// TIA Portal V15.1 export
// export: Created 2024-06-21T08:40:52.1288685Z, ExportSetting WithDefaults, DisplayName Totally Integrated Automation Portal, DisplayVersion V15.1 Update 5, DisplayName TIA Portal Openness, DisplayVersion V15.1 Update 5, DisplayName SINAMICS Startdrive Advanced, DisplayVersion V15.1, DisplayName G130, G150, S120, S150, SINAMICS MV, S210, DisplayVersion V15.1, DisplayName G110M, G120, G120C, G120D, G120P, DisplayVersion V15.1, DisplayName STEP 7 Professional, DisplayVersion V15.1 Update 5, DisplayName STEP 7 Safety, DisplayVersion V15.1, DisplayName WinCC Professional, DisplayVersion V15.1 Update 5, DisplayName SIMATIC Visualization Architect, DisplayVersion V15.1
FUNCTION "F209210ZS01Output" : Void   // FC7012, F_FBD
TITLE = Safety Inputs ZMProc / Safety Outputs 209210ZS01
{ S7_Optimized_Access := 'TRUE' }
VERSION : 0.1
// stored: AutoNumber false, IsIECCheckEnabled false, UDAEnableTagReadback false
BEGIN

REGION Network 1: **** --------------------- Infeed Roller // 210CR21 --------------------- ****
END_REGION

REGION Network 2: **** 8 - Outputs **** 209000AK03M1-UE130 Power OFF - 210CR21M1
   // SEW Drive Power OFF
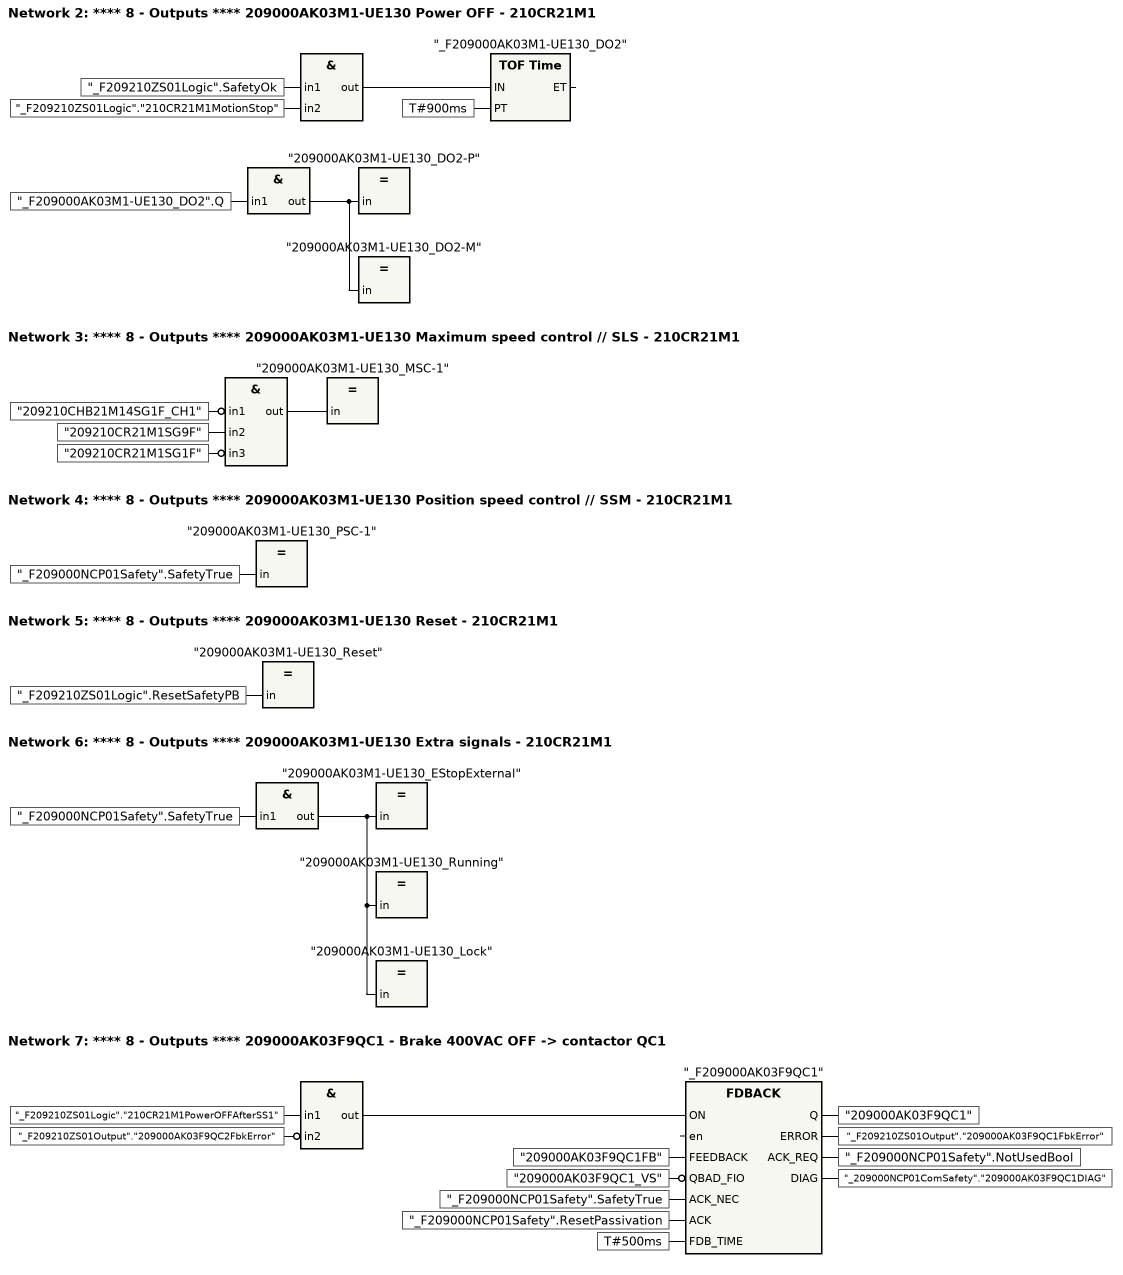
   "_F209000AK03M1-UE130_DO2".TOF(IN := "_F209210ZS01Logic".SafetyOk AND "_F209210ZS01Logic"."210CR21M1MotionStop",
                           PT := T#900ms);
   "209000AK03M1-UE130_DO2-P" := "_F209000AK03M1-UE130_DO2".Q;
   "209000AK03M1-UE130_DO2-M" := "_F209000AK03M1-UE130_DO2".Q;
END_REGION

REGION Network 3: **** 8 - Outputs **** 209000AK03M1-UE130 Maximum speed control // SLS - 210CR21M1
   // SEW Drive Maximum speed control
   "209000AK03M1-UE130_MSC-1" := NOT "209210CHB21M14SG1F_CH1" AND "209210CR21M1SG9F" AND NOT "209210CR21M1SG1F";
END_REGION

REGION Network 4: **** 8 - Outputs **** 209000AK03M1-UE130 Position speed control // SSM - 210CR21M1
   "209000AK03M1-UE130_PSC-1" := "_F209000NCP01Safety".SafetyTrue;
END_REGION

REGION Network 5: **** 8 - Outputs **** 209000AK03M1-UE130 Reset - 210CR21M1
   // SEW Drive Reset
   "209000AK03M1-UE130_Reset" := "_F209210ZS01Logic".ResetSafetyPB;
END_REGION

REGION Network 6: **** 8 - Outputs **** 209000AK03M1-UE130 Extra signals - 210CR21M1
   // SEW Drive Extra signals
   "209000AK03M1-UE130_EStopExternal" := "_F209000NCP01Safety".SafetyTrue;
   "209000AK03M1-UE130_Running" := "_F209000NCP01Safety".SafetyTrue;
   "209000AK03M1-UE130_Lock" := "_F209000NCP01Safety".SafetyTrue;
END_REGION

REGION Network 7: **** 8 - Outputs **** 209000AK03F9QC1 - Brake 400VAC OFF -> contactor QC1
   // Brake 400VAC OFF
   "_F209000AK03F9QC1"(ON := "_F209210ZS01Logic"."210CR21M1PowerOFFAfterSS1" AND NOT "_F209210ZS01Output"."209000AK03F9QC2FbkError",   // FDBACK
                       FEEDBACK := "209000AK03F9QC1FB",
                       QBAD_FIO := NOT "209000AK03F9QC1_VS",
                       ACK_NEC := "_F209000NCP01Safety".SafetyTrue,
                       ACK := "_F209000NCP01Safety".ResetPassivation,
                       FDB_TIME := T#500ms,
                       Q => "209000AK03F9QC1",
                       ERROR => "_F209210ZS01Output"."209000AK03F9QC1FbkError",
                       ACK_REQ => "_F209000NCP01Safety".NotUsedBool,
                       DIAG => "_209000NCP01ComSafety"."209000AK03F9QC1DIAG");
END_REGION

REGION Network 8: **** 8 - Outputs **** 209000AK03F9QC2 - Brake 400VAC OFF -> contactor QC2
   // Brake 400VAC OFF
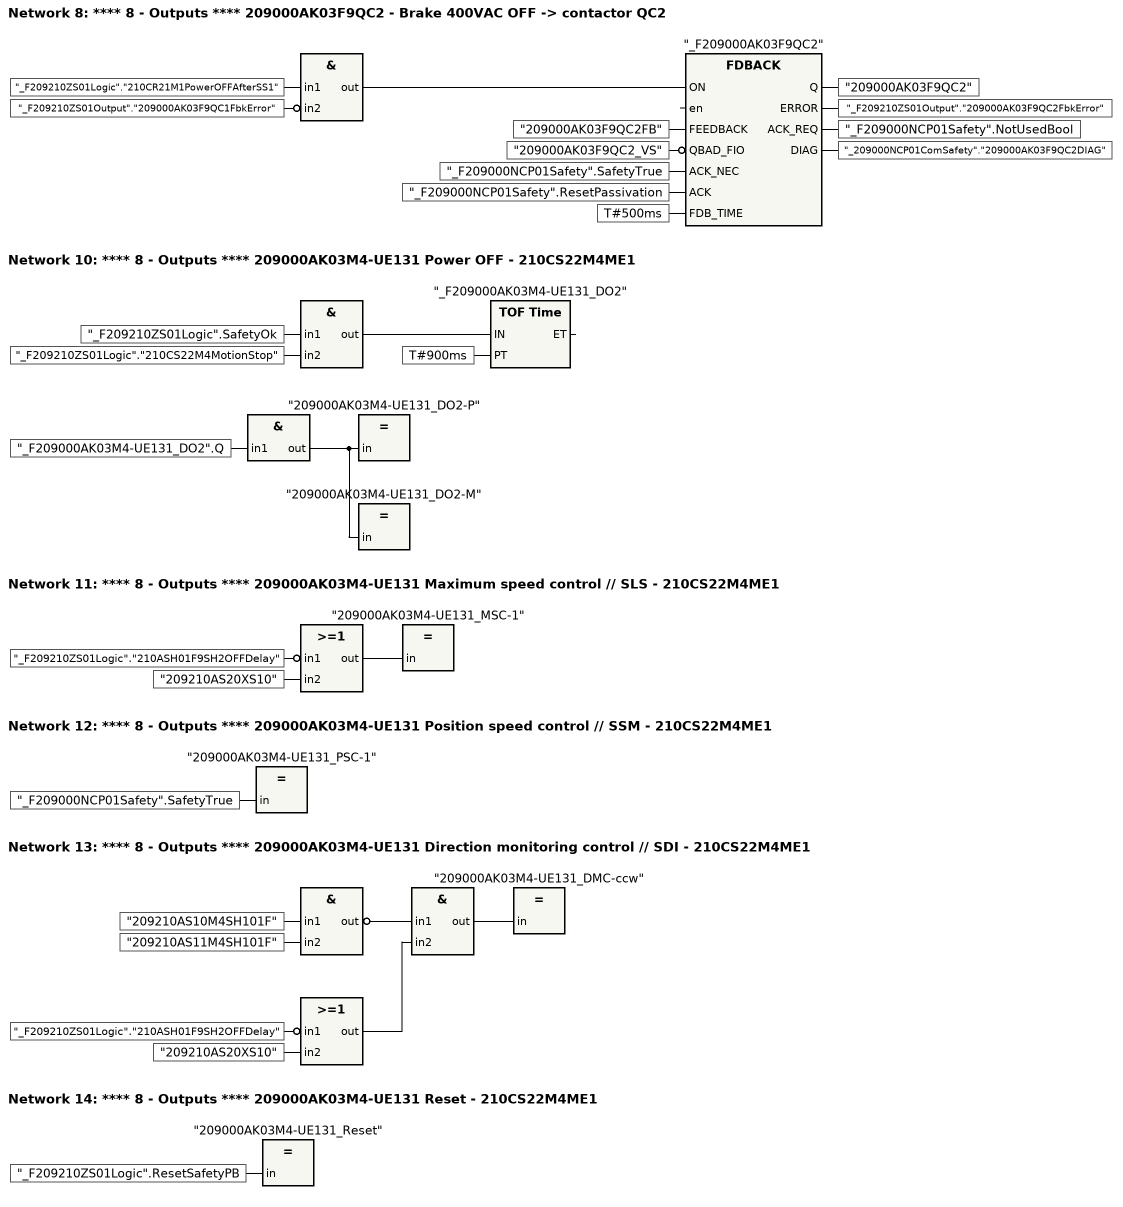
   "_F209000AK03F9QC2"(ON := "_F209210ZS01Logic"."210CR21M1PowerOFFAfterSS1" AND NOT "_F209210ZS01Output"."209000AK03F9QC1FbkError",   // FDBACK
                       FEEDBACK := "209000AK03F9QC2FB",
                       QBAD_FIO := NOT "209000AK03F9QC2_VS",
                       ACK_NEC := "_F209000NCP01Safety".SafetyTrue,
                       ACK := "_F209000NCP01Safety".ResetPassivation,
                       FDB_TIME := T#500ms,
                       Q => "209000AK03F9QC2",
                       ERROR => "_F209210ZS01Output"."209000AK03F9QC2FbkError",
                       ACK_REQ => "_F209000NCP01Safety".NotUsedBool,
                       DIAG => "_209000NCP01ComSafety"."209000AK03F9QC2DIAG");
END_REGION

REGION Network 9: **** --------------------- Slat Conveyor // 210CS22 --------------------- ****
END_REGION

REGION Network 10: **** 8 - Outputs **** 209000AK03M4-UE131 Power OFF - 210CS22M4ME1
   // SEW Drive Power OFF
   "_F209000AK03M4-UE131_DO2".TOF(IN := "_F209210ZS01Logic".SafetyOk AND "_F209210ZS01Logic"."210CS22M4MotionStop",
                           PT := T#900ms);
   "209000AK03M4-UE131_DO2-P" := "_F209000AK03M4-UE131_DO2".Q;
   "209000AK03M4-UE131_DO2-M" := "_F209000AK03M4-UE131_DO2".Q;
END_REGION

REGION Network 11: **** 8 - Outputs **** 209000AK03M4-UE131 Maximum speed control // SLS - 210CS22M4ME1
   // SEW Drive Maximum speed control
   "209000AK03M4-UE131_MSC-1" := NOT "_F209210ZS01Logic"."210ASH01F9SH2OFFDelay" OR "209210AS20XS10";
END_REGION

REGION Network 12: **** 8 - Outputs **** 209000AK03M4-UE131 Position speed control // SSM - 210CS22M4ME1
   "209000AK03M4-UE131_PSC-1" := "_F209000NCP01Safety".SafetyTrue;
END_REGION

REGION Network 13: **** 8 - Outputs **** 209000AK03M4-UE131 Direction monitoring control // SDI - 210CS22M4ME1
   "209000AK03M4-UE131_DMC-ccw" := NOT ("209210AS10M4SH101F" AND "209210AS11M4SH101F") AND (NOT "_F209210ZS01Logic"."210ASH01F9SH2OFFDelay" OR "209210AS20XS10");
END_REGION

REGION Network 14: **** 8 - Outputs **** 209000AK03M4-UE131 Reset - 210CS22M4ME1
   // SEW Drive Reset
   "209000AK03M4-UE131_Reset" := "_F209210ZS01Logic".ResetSafetyPB;
END_REGION

REGION Network 15: **** 8 - Outputs **** 209000AK03M4-UE131 Extra signals - 210CS22M4ME1
   // SEW Drive Extra signals
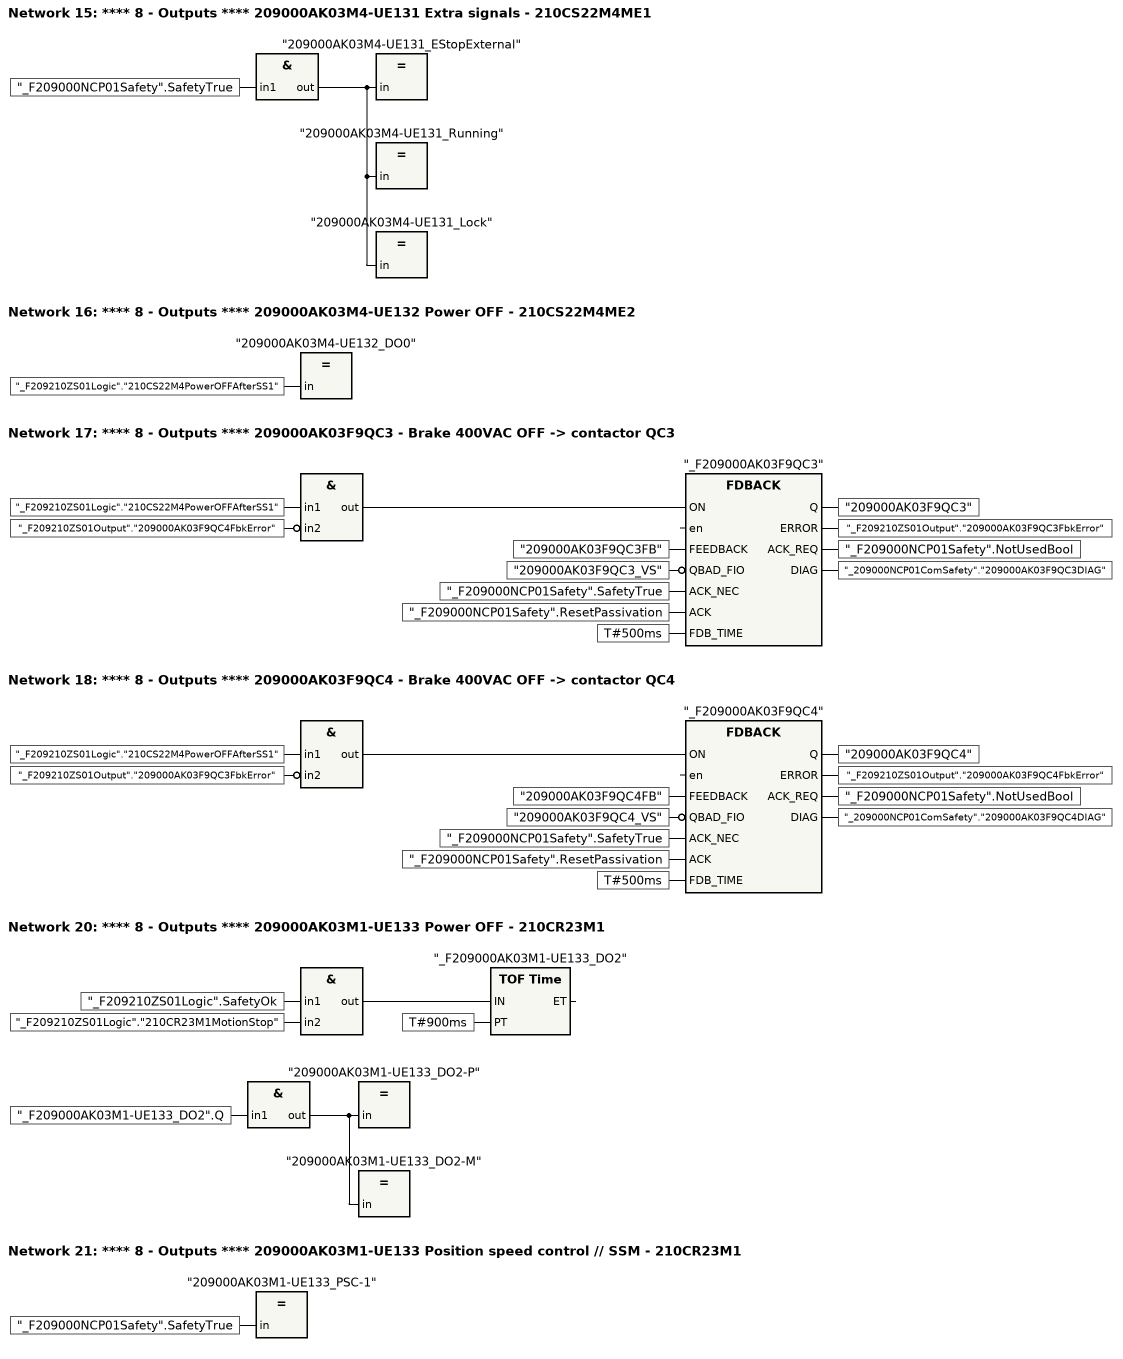
   "209000AK03M4-UE131_EStopExternal" := "_F209000NCP01Safety".SafetyTrue;
   "209000AK03M4-UE131_Running" := "_F209000NCP01Safety".SafetyTrue;
   "209000AK03M4-UE131_Lock" := "_F209000NCP01Safety".SafetyTrue;
END_REGION

REGION Network 16: **** 8 - Outputs **** 209000AK03M4-UE132 Power OFF - 210CS22M4ME2
   // SEW Drive Power OFF
   "209000AK03M4-UE132_DO0" := "_F209210ZS01Logic"."210CS22M4PowerOFFAfterSS1";
END_REGION

REGION Network 17: **** 8 - Outputs **** 209000AK03F9QC3 - Brake 400VAC OFF -> contactor QC3
   // Brake 400VAC OFF
   "_F209000AK03F9QC3"(ON := "_F209210ZS01Logic"."210CS22M4PowerOFFAfterSS1" AND NOT "_F209210ZS01Output"."209000AK03F9QC4FbkError",   // FDBACK
                       FEEDBACK := "209000AK03F9QC3FB",
                       QBAD_FIO := NOT "209000AK03F9QC3_VS",
                       ACK_NEC := "_F209000NCP01Safety".SafetyTrue,
                       ACK := "_F209000NCP01Safety".ResetPassivation,
                       FDB_TIME := T#500ms,
                       Q => "209000AK03F9QC3",
                       ERROR => "_F209210ZS01Output"."209000AK03F9QC3FbkError",
                       ACK_REQ => "_F209000NCP01Safety".NotUsedBool,
                       DIAG => "_209000NCP01ComSafety"."209000AK03F9QC3DIAG");
END_REGION

REGION Network 18: **** 8 - Outputs **** 209000AK03F9QC4 - Brake 400VAC OFF -> contactor QC4
   // Brake 400VAC OFF
   "_F209000AK03F9QC4"(ON := "_F209210ZS01Logic"."210CS22M4PowerOFFAfterSS1" AND NOT "_F209210ZS01Output"."209000AK03F9QC3FbkError",   // FDBACK
                       FEEDBACK := "209000AK03F9QC4FB",
                       QBAD_FIO := NOT "209000AK03F9QC4_VS",
                       ACK_NEC := "_F209000NCP01Safety".SafetyTrue,
                       ACK := "_F209000NCP01Safety".ResetPassivation,
                       FDB_TIME := T#500ms,
                       Q => "209000AK03F9QC4",
                       ERROR => "_F209210ZS01Output"."209000AK03F9QC4FbkError",
                       ACK_REQ => "_F209000NCP01Safety".NotUsedBool,
                       DIAG => "_209000NCP01ComSafety"."209000AK03F9QC4DIAG");
END_REGION

REGION Network 19: **** --------------------- Outfeed Roller // 210CR23 --------------------- ****
END_REGION

REGION Network 20: **** 8 - Outputs **** 209000AK03M1-UE133 Power OFF - 210CR23M1
   // SEW Drive Power OFF
   "_F209000AK03M1-UE133_DO2".TOF(IN := "_F209210ZS01Logic".SafetyOk AND "_F209210ZS01Logic"."210CR23M1MotionStop",
                           PT := T#900ms);
   "209000AK03M1-UE133_DO2-P" := "_F209000AK03M1-UE133_DO2".Q;
   "209000AK03M1-UE133_DO2-M" := "_F209000AK03M1-UE133_DO2".Q;
END_REGION

REGION Network 21: **** 8 - Outputs **** 209000AK03M1-UE133 Position speed control // SSM - 210CR23M1
   "209000AK03M1-UE133_PSC-1" := "_F209000NCP01Safety".SafetyTrue;
END_REGION

REGION Network 22: **** 8 - Outputs **** 209000AK03M1-UE133 Direction monitoring control // SDI - 210CR23M1
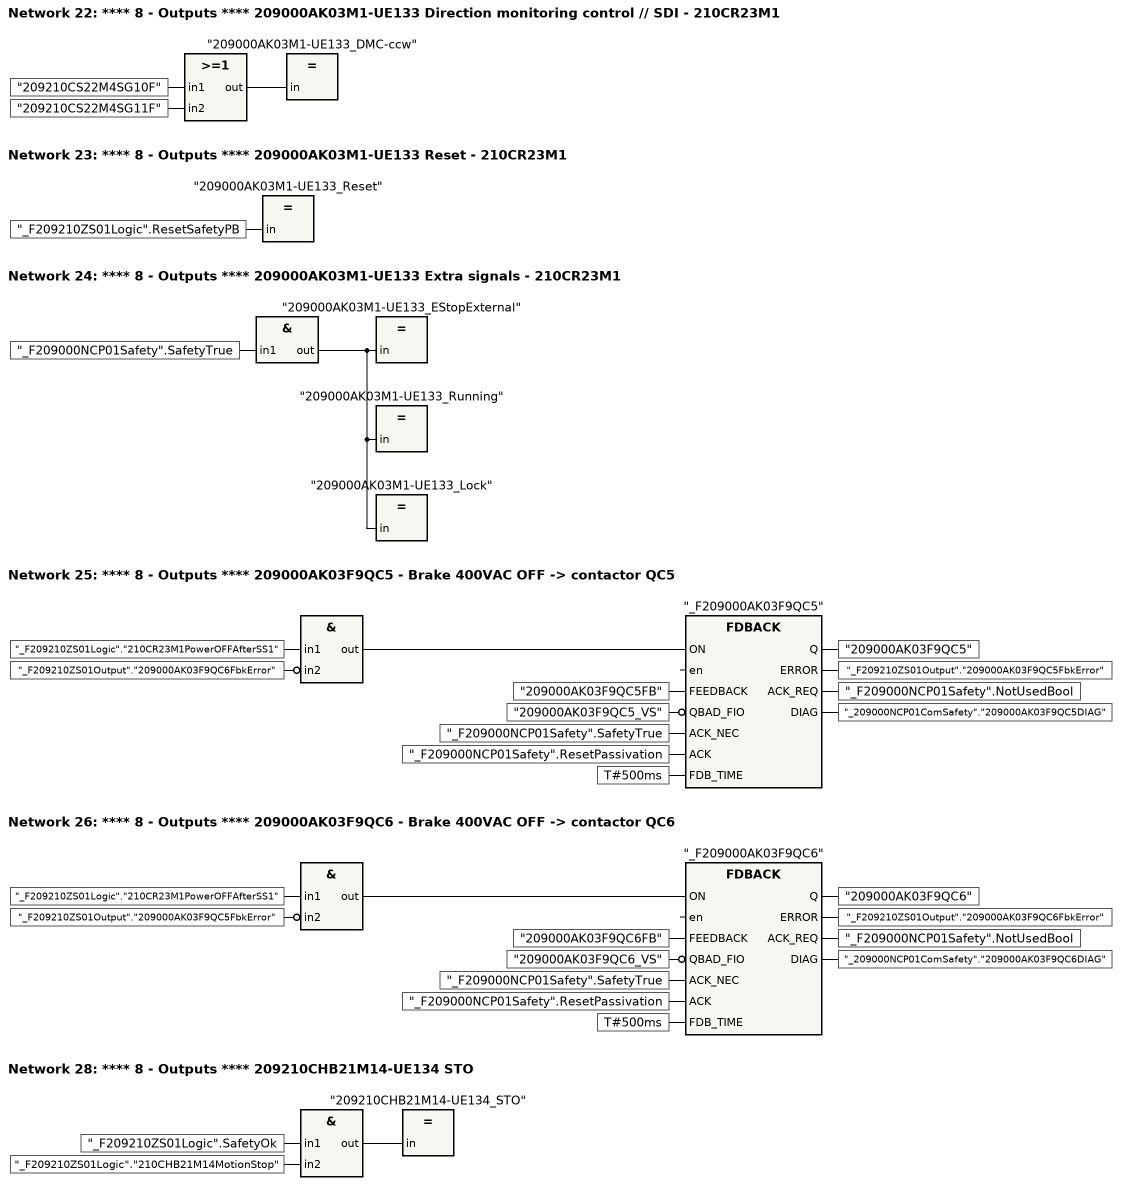
   "209000AK03M1-UE133_DMC-ccw" := "209210CS22M4SG10F" OR "209210CS22M4SG11F";
END_REGION

REGION Network 23: **** 8 - Outputs **** 209000AK03M1-UE133 Reset - 210CR23M1
   // SEW Drive Reset
   "209000AK03M1-UE133_Reset" := "_F209210ZS01Logic".ResetSafetyPB;
END_REGION

REGION Network 24: **** 8 - Outputs **** 209000AK03M1-UE133 Extra signals - 210CR23M1
   // SEW Drive Extra signals
   "209000AK03M1-UE133_EStopExternal" := "_F209000NCP01Safety".SafetyTrue;
   "209000AK03M1-UE133_Running" := "_F209000NCP01Safety".SafetyTrue;
   "209000AK03M1-UE133_Lock" := "_F209000NCP01Safety".SafetyTrue;
END_REGION

REGION Network 25: **** 8 - Outputs **** 209000AK03F9QC5 - Brake 400VAC OFF -> contactor QC5
   // Brake 400VAC OFF
   "_F209000AK03F9QC5"(ON := "_F209210ZS01Logic"."210CR23M1PowerOFFAfterSS1" AND NOT "_F209210ZS01Output"."209000AK03F9QC6FbkError",   // FDBACK
                       FEEDBACK := "209000AK03F9QC5FB",
                       QBAD_FIO := NOT "209000AK03F9QC5_VS",
                       ACK_NEC := "_F209000NCP01Safety".SafetyTrue,
                       ACK := "_F209000NCP01Safety".ResetPassivation,
                       FDB_TIME := T#500ms,
                       Q => "209000AK03F9QC5",
                       ERROR => "_F209210ZS01Output"."209000AK03F9QC5FbkError",
                       ACK_REQ => "_F209000NCP01Safety".NotUsedBool,
                       DIAG => "_209000NCP01ComSafety"."209000AK03F9QC5DIAG");
END_REGION

REGION Network 26: **** 8 - Outputs **** 209000AK03F9QC6 - Brake 400VAC OFF -> contactor QC6
   // Brake 400VAC OFF
   "_F209000AK03F9QC6"(ON := "_F209210ZS01Logic"."210CR23M1PowerOFFAfterSS1" AND NOT "_F209210ZS01Output"."209000AK03F9QC5FbkError",   // FDBACK
                       FEEDBACK := "209000AK03F9QC6FB",
                       QBAD_FIO := NOT "209000AK03F9QC6_VS",
                       ACK_NEC := "_F209000NCP01Safety".SafetyTrue,
                       ACK := "_F209000NCP01Safety".ResetPassivation,
                       FDB_TIME := T#500ms,
                       Q => "209000AK03F9QC6",
                       ERROR => "_F209210ZS01Output"."209000AK03F9QC6FbkError",
                       ACK_REQ => "_F209000NCP01Safety".NotUsedBool,
                       DIAG => "_209000NCP01ComSafety"."209000AK03F9QC6DIAG");
END_REGION

REGION Network 27: **** --------------------- Hold Back // 210CHB21 --------------------- ****
END_REGION

REGION Network 28: **** 8 - Outputs **** 209210CHB21M14-UE134 STO
   // SEW Drive STO
   "209210CHB21M14-UE134_STO" := "_F209210ZS01Logic".SafetyOk AND "_F209210ZS01Logic"."210CHB21M14MotionStop";
END_REGION
END_FUNCTION
